(* IEC 61131-3 sources: AutomationStudio/KomoraCieplna/KomCont, 3 files *)

(* ---- Types.typ ---- *)
TYPE
	ModeTyp :
		(
		NONE := 0, (* Nie wybrany algorytm *)
		MANUAL := 1, (*Sterowanie ręczne*)
		ONOFF := 2, (* Algorytm dwustawny *)
		PID := 3, (* ALgorytm PID *)
		FUZZY := 4, (* Algorytm rozmyty *)
		ADRC := 5, (* Algortym adaptacyjny *)
		DEADBEAT :=6 (* Algorytm cyfrowy dead beat *)
		);
	KomoraTyp : 	STRUCT
		aoHeater : INT; (* Wysterowanie grzałki *)
		aoFan : INT; (* Wysterowanie wentylatora *)
		aiTemperature : INT; (* Pomiar temperatury -> PT1000 *)
		uiHeater : REAL; (* Wysterowanie grzałki -> GUI [%]*)
		uiFan : REAL; (* Wysterowanie wentylatora -> GUI [%] *)
		uiTemperature : REAL; (* Pomiar temperatury -> PT1000 -> GUI [oC] *)
		Heater : AnalogActuatorTyp;
		Fan : AnalogActuatorTyp;
		Temperature : AnalogSensorTyp;
		TemperatureOutSide : AnalogSensorTyp;
	END_STRUCT;

	sKomoraParTyp : STRUCT
		k : REAL; (* Wzmocnienie części proporcjonalnej - skalowanie strumień ciepła - wartość temperatury*)
		T1 : REAL; (* Stała czasowa bezwładności [s -default, min, h] *)
		T2 : REAL; (* Stała czasowa bezwładności [s -default, min, h] *)
	END_STRUCT;

	AnalogActuatorTyp : 	STRUCT
		aoValue : INT;
		uiStatus : USINT;
		uiValue : REAL;
	END_STRUCT;
	AnalogSensorTyp : 	STRUCT
		aiValue : INT;
		uiStatus : USINT;
		uiValue : REAL;
	END_STRUCT;
	OperatorTyp : 	STRUCT
		Heater : AnalogActuatorTyp; (* Do sterowania ręcznego grzaniem -> suwak i pole num *)
		Fan : AnalogActuatorTyp; (* Do sterowania ręcznego wentylowaniem -> suwak i pole num *)
		diStart : BOOL; (* Przycisk Start - inicjowanie pracy systemu *)
		diStop : BOOL; (* Przycisk Stop - zatrzymywanie pracy systemu *)
		diEStop : BOOL:= TRUE; (* Przycisk EStop - zatrzymywanie pracy systemu Emergency Switch*)
		doSystemAktywny : BOOL; (* Lampka system aktywny *)
		uiStart : BOOL; (* Kontrolka Start - inicjowanie pracy systemu - GUI*)
		uiStop : BOOL; (* Kontrolka Stop - zatrzymywanie pracy systemu - GUI*)
		uiSystemAktywny : BOOL; (* Kontrolka system aktywny - GUI*)
		diReset : BOOL; (* Przycisk kasowania awarii *)
		doAlarm : BOOL; (* Lampka awaria *)
		uiReset : BOOL; (* Kontrolka-dotyk kasowania awarii - GUI*)
		uiAlarm : BOOL; (* Kontrolka - Lampka awaria - GUI*)
		GUI : GUITyp; (* Zmienna złożona do sterowania elementami graficznymi *)
	END_STRUCT;

	GUITyp : STRUCT
		uiEnableSimulation : BOOL:= TRUE; (* Aktywacja symulacji komory cieplnej*)
		uiLockWindow : USINT;
		ShowLayer : LayerTyp;
		Units : UnitTyp;
	END_STRUCT;

	UnitTyp : STRUCT
		uiHeater : USINT;
		uiTemperature : USINT;
	END_STRUCT;

	LayerTyp : STRUCT
		Manual : USINT;
		OnOff : USINT;
		PID : USINT;
	END_STRUCT;

END_TYPE

(* ---- Main.st ---- *)
PROGRAM _INIT
	(* Insert code here *)
	Operator[0].GUI.Units.uiHeater:=1; (* Jednostki wydajności grzałki : 0=int, 1=%,2-volt *)
	Operator[0].GUI.Units.uiTemperature:=1	;(* Jednostki temp : 0=int, 1=oC,2-oF *)
END_PROGRAM

PROGRAM _CYCLIC
	(* Kooperacja z Matlab/Simulink *)
	gTemperaturePV:= Komora[0].Temperature.uiValue;
	gTemperatureSP:= gKomoraPar[0].TemperatureSP;
	gError:= gKomoraPar[0].TemperatureSP - Komora[0].Temperature.uiValue;
	(* Procedura Uruchamiania i zatrzymywania procesu *)

	Operator[0].uiSystemAktywny:= (Operator[0].uiStart OR Operator[0].uiSystemAktywny)	AND
	NOT(Operator[0].uiStop) AND Operator[0].diEStop; (* Aktywacja systemu z priorytetem na Stop *)

	gOperator.Enable:= Operator[0].uiSystemAktywny;//Przekazanie flagi do zmiennej globalnej -> aktywacja OnOff, PID itd

	Komora[0].TemperatureOutSide.uiValue:= INT_TO_REAL(Komora[0].TemperatureOutSide.aiValue); //Temperatura otoczenia

	IF Operator[0].GUI.uiEnableSimulation THEN
		(* Komora symulowana - model PT2 *)
		sKomora[0].Enable:= gOperator.Enable; //System aktywny
		sKomora[0].Gain:= sKomoraPar[0].k; //Wzmocnienie proporcjonalne
		sKomora[0].TimeConstant1:= sKomoraPar[0].T1; //Stała czasowa T1
		sKomora[0].TimeConstant2:= sKomoraPar[0].T2; //Stała czasowa T2
		sKomora[0](); //FUB - function update block
		Komora[0].Temperature.uiValue:= sKomora[0].Out; (* Komora symulowana *)
		sKomora[0].Update:= EDGEPOS(gOperator.Enable); //Wczytanie k, T1, T2 do rejestrów modelu
		gHeaterCV:= sKomora[0].In;
	ELSE
		Komora[0].Temperature.uiValue:= INT_TO_REAL(Komora[0].Temperature.aiValue);(* Komora rzeczywista *)
		gHeaterCV:= INT_TO_REAL(Komora[0].Heater.aoValue);
	END_IF;

	CASE Tryb[0] OF

		NONE:
			Komora[0].Heater.aoValue:= 0; //uiValue -> GUI
			Komora[0].Fan.aoValue:= 0;	//Ręczne sterowanie obiektem
		MANUAL:
			IF Operator[0].GUI.uiEnableSimulation THEN
					sKomora[0].In:= Operator[0].Heater.uiValue; //uiValue -> GUI
					//Komora[0].Fan.aoValue:= REAL_TO_INT(Operator[0].Fan.uiValue);	//Ręczne sterowanie obiektem
				ELSE
					Komora[0].Heater.aoValue:= 	REAL_TO_INT(Operator[0].Heater.uiValue); //uiValue -> GUI
					Komora[0].Fan.aoValue:= REAL_TO_INT(Operator[0].Fan.uiValue);	//Ręczne sterowanie obiektem
				END_IF;

		ONOFF:
				gOnOff.Enable:=Operator[0].uiSystemAktywny;
				IF Operator[0].GUI.uiEnableSimulation THEN
					//Komora[0].Fan.aoValue:= REAL_TO_INT(Operator[0].Fan.uiValue); (* Sterowanie ręczne *)
					sKomora[0].In:= gOnOff.HeaterCV; //Pobieranie sygnału sterującego z OnOff
					gOnOff.TemperaturePV:= Komora[0].Temperature.uiValue;//Wysyłanie sygnału pomiarowego do OnOff
				ELSE
					Komora[0].Fan.aoValue:= REAL_TO_INT(Operator[0].Fan.uiValue); (* Sterowanie ręczne *)
					Komora[0].Heater.aoValue:= 	REAL_TO_INT(gOnOff.HeaterCV); //Pobieranie sygnału sterującego z OnOff
					gOnOff.TemperaturePV:= INT_TO_REAL(Komora[0].Temperature.aiValue);//Wysyłanie sygnału pomiarowego do OnOff
				END_IF;

		PID:
				gPID.Enable:=Operator[0].uiSystemAktywny;
				IF Operator[0].GUI.uiEnableSimulation THEN
					//Komora[0].Fan.aoValue:= REAL_TO_INT(Operator[0].Fan.uiValue); (* Sterowanie ręczne *)
					sKomora[0].In:= gPID.HeaterCV; //Pobieranie sygnału sterującego z PID
					gPID.TemperaturePV:= Komora[0].Temperature.uiValue;//Wysyłanie sygnału pomiarowego do PID
				ELSE
					Komora[0].Fan.aoValue:= REAL_TO_INT(Operator[0].Fan.uiValue); (* Sterowanie ręczne *)
					Komora[0].Heater.aoValue:= 	REAL_TO_INT(gPID.HeaterCV); //Pobieranie sygnału sterującego z PID
					gPID.TemperaturePV:= INT_TO_REAL(Komora[0].Temperature.aiValue);//Wysyłanie sygnału pomiarowego do PID
				END_IF;
		FUZZY:
			Komora[0].Fan.aoValue:= REAL_TO_INT(Operator[0].Fan.uiValue);

		ADRC:
			Komora[0].Fan.aoValue:= REAL_TO_INT(Operator[0].Fan.uiValue);

		DEADBEAT:
			Komora[0].Fan.aoValue:= REAL_TO_INT(Operator[0].Fan.uiValue);

	END_CASE;

END_PROGRAM

PROGRAM _EXIT
	(* Insert code here *)

END_PROGRAM

(* ---- Variables.var ---- *)
VAR
	Komora : ARRAY[0..1] OF KomoraTyp; (* Struktura obiektu sterowania *)
	sKomora : ARRAY[0..1] OF MTBasicsPT2; (* Struktura modelu obiektu PT2 *)
	Operator : ARRAY[0..1] OF OperatorTyp; (* Struktura obsługi obiektu sterowania *)
	Tryb : ARRAY[0..1] OF ModeTyp; (* Struktura algorytmów sterowania *)
	Delay : ARRAY[0..10] OF TON; (* zegarki *)
	LiczMinMax : ARRAY[0..10] OF LCRMinMax; (* Funkcja liczenia min i max *)
	fTempOnOff : BOOL; (* flaga do wyznaczenia wykresuy PU *)
	fCzasStartStop : BOOL; (* flaga pomiaru czasu - start/stop zegara*)
END_VAR

VAR RETAIN
	sKomoraPar : ARRAY[0..1] OF sKomoraParTyp; (* Parametry obiektu do wpisywania z GUI *)

END_VAR
